SUBAPPLICATION Uebung_127 (* Übung zu ISOBUS Send Message Cyclic (ohne CB) *)
  (* Standard: 61499-2; Description: Copyright (c) 2025 Meisterschulen am Ostbahnhof This program and the accompanying materials are made available under the terms of the Eclipse Public License 2.0 which is available at https://www.eclipse.org/legal/epl-2.0/ SPDX-License-Identifier: EPL-2.0 *)
  (* Version 1.0, 2023-10-23, Franz Höpfinger, Meisterschulen am Ostbahnhof *)
  PACKAGE Uebungen;
  IMPORT isobus::pgn::ISOUSERHOME_e::network;
  IMPORT isobus::pgn::ISO_CAN_NODE::NODE1;
  IMPORT logiBUS::io::DI::logiBUS_DI::Input_I1;
  IMPORT logiBUS::io::DI::logiBUS_DI_Events::BUTTON_SINGLE_CLICK;
  IMPORT Uebungen::const::Uebung_120_129::Filter::VT_ADD;
  IMPORT Uebungen::const::Uebung_120_129::Filter::VT_FLT;
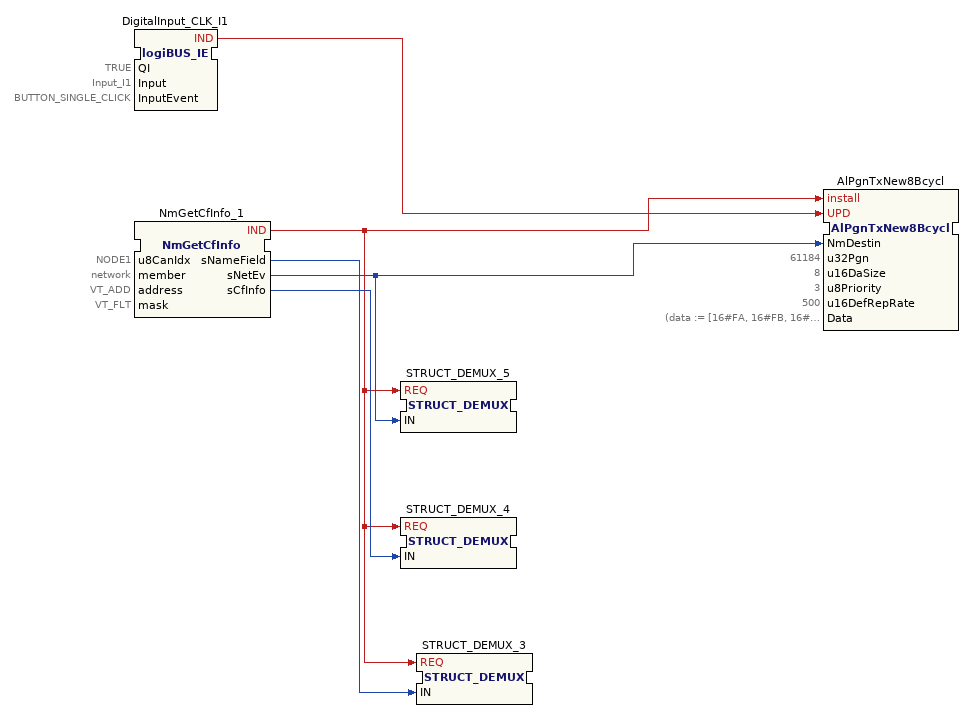
  FBS
    STRUCT_DEMUX_3 : eclipse4diac::convert::STRUCT_DEMUX; {SET_ATTRIBUTE(StructuredType, isobus::pgn::NAMEFIELD_T)}
    NmGetCfInfo_1 : isobus::pgn::NmGetCfInfo(u8CanIdx := NODE1, member := network, address := VT_ADD, mask := VT_FLT);
    STRUCT_DEMUX_4 : eclipse4diac::convert::STRUCT_DEMUX; {SET_ATTRIBUTE(StructuredType, isobus::pgn::CF_INFO_T)}
    STRUCT_DEMUX_5 : eclipse4diac::convert::STRUCT_DEMUX; {SET_ATTRIBUTE(StructuredType, isobus::pgn::ISONETEVENT_T)}
    AlPgnTxNew8Bcycl : isobus::pgn::tx::AlPgnTxNew8Bcycl(u32Pgn := 61184, u16DaSize := 8, u8Priority := 3, u16DefRepRate := 500, Data := (data := [16#FA, 16#FB, 16#FC, 16#FD, 16#FE, 16#FF, 16#F1, 16#F2]));
    DigitalInput_CLK_I1 : logiBUS::io::DI::logiBUS_IE(QI := TRUE, Input := Input_I1, InputEvent := BUTTON_SINGLE_CLICK);
  END_FBS
  EVENT_CONNECTIONS
    NmGetCfInfo_1.IND TO STRUCT_DEMUX_3.REQ;
    NmGetCfInfo_1.IND TO STRUCT_DEMUX_4.REQ;
    NmGetCfInfo_1.IND TO STRUCT_DEMUX_5.REQ;
    NmGetCfInfo_1.IND TO AlPgnTxNew8Bcycl.install;
    DigitalInput_CLK_I1.IND TO AlPgnTxNew8Bcycl.UPD;
  END_CONNECTIONS
  DATA_CONNECTIONS
    NmGetCfInfo_1.sNameField TO STRUCT_DEMUX_3.IN;
    NmGetCfInfo_1.sNetEv TO STRUCT_DEMUX_5.IN;
    NmGetCfInfo_1.sCfInfo TO STRUCT_DEMUX_4.IN;
    NmGetCfInfo_1.sNetEv TO AlPgnTxNew8Bcycl.NmDestin;
  END_CONNECTIONS
END_SUBAPPLICATION
